// TIA Portal V17 export
// export: Created 2023-04-03T06:31:42.3399375Z, ExportSetting WithDefaults, DisplayName Totally Integrated Automation Portal, DisplayVersion V17 Update 4, DisplayName TIA Portal Openness, DisplayVersion V17 Update 4, DisplayName TIA Portal Version Control Interface, DisplayVersion V17, DisplayName STEP 7 Professional, DisplayVersion V17 Update 4, DisplayName STEP 7 Safety, DisplayVersion V17, DisplayName WinCC Professional, DisplayVersion V17 Update 4
TYPE "W_PE_Block3"
// stored: IsFailsafeCompliant false
   STRUCT
      "G15.1.2_Banks_Enabled" : Word;   // 1
      "G8.1.3a_Pac_Reference_1" : Real;   // 94
      "G8.1.3b_Pac_Reference_2" : Real;   // 95
   END_STRUCT;
END_TYPE
